FUNCTION F_factorial : ULINT
VAR_INPUT
	n : ULINT;
END_VAR
VAR
	tempFact : ULINT;
	i : ULINT;
END_VAR

tempFact := 1;
FOR i := 1 TO n BY 1 DO
	tempFact := i * tempFact;
END_FOR
F_factorial := tempFact;

END_FUNCTION

(* stored: Version 1.1.0.1, ProductVersion 3.1.4024.12
   POU F_factorial: Id {f87b3d5b-dbf2-4dae-adf5-c11145cff916}, SpecialFunc None *)
